// TIA Portal V18 export
ORGANIZATION_BLOCK "Main"   // OB1, LAD, ProgramCycle
TITLE = "Main Program Sweep (Cycle)"
{ S7_Optimized_Access := 'TRUE' }
// stored: SetENOAutomatically false
   VAR_INPUT
      Initial_Call : Bool;   // Initial call of this OB
      Remanence : Bool;   // =True, if remanent data are available
   END_VAR
BEGIN

REGION Network 1: 00_Diagnostic PB
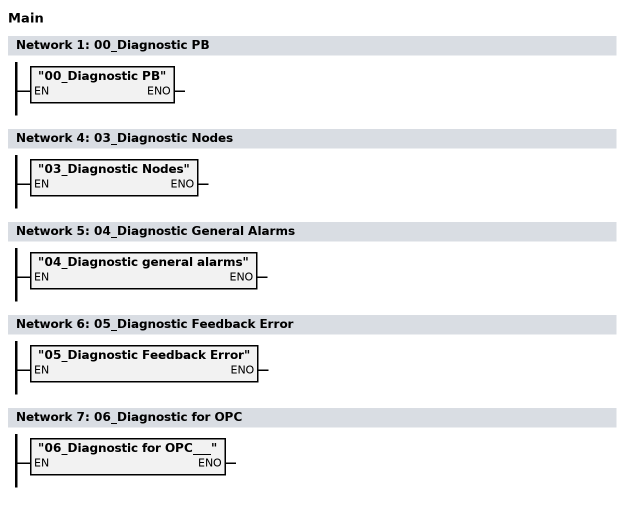
   RUNG wire#powerrail
      "00_Diagnostic PB"()
   END_RUNG
   // the same network as SCL:
   "00_Diagnostic PB"();
END_REGION

REGION Network 2: 01_Diagnostic Status
END_REGION

REGION Network 3: 02_Diagnostic Profinet
END_REGION

REGION Network 4: 03_Diagnostic Nodes
   RUNG wire#powerrail
      "03_Diagnostic Nodes"()
   END_RUNG
   // the same network as SCL:
   "03_Diagnostic Nodes"();
END_REGION

REGION Network 5: 04_Diagnostic General Alarms
   RUNG wire#powerrail
      "04_Diagnostic general alarms"()
   END_RUNG
   // the same network as SCL:
   "04_Diagnostic general alarms"();
END_REGION

REGION Network 6: 05_Diagnostic Feedback Error
   RUNG wire#powerrail
      "05_Diagnostic Feedback Error"()
   END_RUNG
   // the same network as SCL:
   "05_Diagnostic Feedback Error"();
END_REGION

REGION Network 7: 06_Diagnostic for OPC
   RUNG wire#powerrail
      "06_Diagnostic for OPC___"()
   END_RUNG
   // the same network as SCL:
   "06_Diagnostic for OPC___"();
END_REGION
END_ORGANIZATION_BLOCK
